// TIA Portal V20 export
// export: Created 2025-12-01T14:57:26.4932123Z, ExportSetting None, DisplayName Totally Integrated Automation Portal, DisplayVersion V20 Update 3, DisplayName TIA Portal Openness, DisplayVersion V20 Update 3, DisplayName TIA Portal Version Control Interface, DisplayVersion V20 Update 3, DisplayName STEP 7 Professional, DisplayVersion V20 Update 3, DisplayName STEP 7 Safety, DisplayVersion V20 Update 2, DisplayName WinCC Basic/Comfort/Advanced, DisplayVersion V20 Update 3, DisplayName WinCC Professional, DisplayVersion V20 Update 3, DisplayName WinCC Unified, DisplayVersion V20 Update 3
DATA_BLOCK "DB602_ElementosQuimarox"   // DB602
{ S7_Optimized_Access := 'FALSE' }
// stored: AutoNumber false
   VAR RETAIN
      Quimarox : Array[1.."CTE_MaxNumQuimarox"] of Struct
         Elementos { S7_SetPoint := 'True'} : Array[1.."CTE_MaxNumElementos"] of "CBS_Elemento";
      END_STRUCT;
   END_VAR
BEGIN
   Quimarox[1].Elementos[1].posicion_real_elemento := 700.0;
   Quimarox[1].Elementos[2].posicion_real_elemento := 7700.0;
   Quimarox[1].Elementos[3].posicion_real_elemento := 14890.0;
   Quimarox[1].Elementos[4].posicion_real_elemento := 18000.0;
   Quimarox[1].Elementos[5].posicion_real_elemento := 6870.7;
   Quimarox[1].Elementos[1..5].ventana_minima := 50;
   Quimarox[1].Elementos[1].ventana_maxima := 1400;
   Quimarox[1].Elementos[2..5].ventana_maxima := 1550;
   Quimarox[1].Elementos[6..50].Numero_carrier := 11;
   Quimarox[1].Elementos[6..34].Avance_carrier := 1069;
   Quimarox[1].Elementos[35..47].Avance_carrier := 1079;
   Quimarox[1].Elementos[48..50].Avance_carrier := 1083;
END_DATA_BLOCK
